{attribute 'GeneratedUsingTerminal: EL2911-0000-0016'}
{attribute addProperty BoxType "EL2911-0000-0016"}
{attribute addProperty Id "Fieldvoltage_UnderrangeAT %I*BOOL1Fieldvoltage_OverrangeAT %I*BOOL1"}
{attribute addProperty CRC "2647114569"}
{attribute addProperty Size "2"}
TYPE FIELDVOLTAGE_Field_Voltage_Status_9DC7C349 EXTENDS InputBase_8311D824 :
STRUCT
	{attribute addProperty Name "Fieldvoltage_Underrange"}
	Fieldvoltage_Underrange AT %I* : BOOL;
	{attribute addProperty Name "Fieldvoltage_Overrange"}
	Fieldvoltage_Overrange AT %I* : BOOL;
END_STRUCT
END_TYPE

(* stored: Version 1.2.0.0, ProductVersion 3.1.4024.9
   DUT FIELDVOLTAGE_Field_Voltage_Status_9DC7C349: Id {0c941130-890f-49bc-8ef1-9902bce57afd} *)
